Staubli VAL3: FwdBoxType.pgx

public program FwdBoxType()
begin
    if nBoxType<2
    nBoxType=nBoxType+1
  else
    nBoxType=1
    endIf
end
